FUNCTION_BLOCK Physical_Plant_SIMULATION (* Composite Function Block Type *)
  (* Standard: 61499-2 *)
  (* Version 0.0, 12/12/2023, Cheyan, Schneider Electric, template *)
  PACKAGE Main;
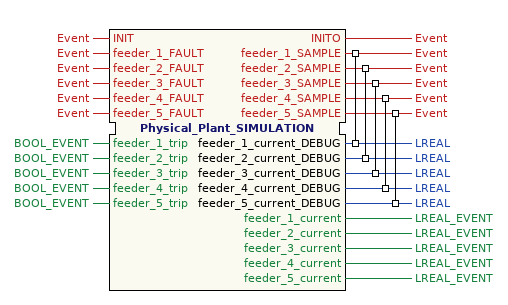
  EVENT_INPUT
    INIT; (* Initialization Request *)
    feeder_1_FAULT;
    feeder_2_FAULT;
    feeder_3_FAULT;
    feeder_4_FAULT;
    feeder_5_FAULT;
  END_EVENT
  EVENT_OUTPUT
    INITO; (* Initialization Confirm *)
    feeder_1_SAMPLE WITH feeder_1_current_DEBUG;
    feeder_2_SAMPLE WITH feeder_2_current_DEBUG;
    feeder_3_SAMPLE WITH feeder_3_current_DEBUG;
    feeder_4_SAMPLE WITH feeder_4_current_DEBUG;
    feeder_5_SAMPLE WITH feeder_5_current_DEBUG;
  END_EVENT
  VAR_OUTPUT
    feeder_1_current_DEBUG : LREAL; (* Output event qualifier *)
    feeder_2_current_DEBUG : LREAL; (* Output event qualifier *)
    feeder_3_current_DEBUG : LREAL; (* Output event qualifier *)
    feeder_4_current_DEBUG : LREAL; (* Output event qualifier *)
    feeder_5_current_DEBUG : LREAL; (* Output event qualifier *)
  END_VAR
  SOCKETS
    feeder_1_trip : BOOL_EVENT;
    feeder_2_trip : BOOL_EVENT;
    feeder_3_trip : BOOL_EVENT;
    feeder_4_trip : BOOL_EVENT;
    feeder_5_trip : BOOL_EVENT;
  END_SOCKETS
  PLUGS
    feeder_1_current : LREAL_EVENT;
    feeder_2_current : LREAL_EVENT;
    feeder_3_current : LREAL_EVENT;
    feeder_4_current : LREAL_EVENT;
    feeder_5_current : LREAL_EVENT;
  END_PLUGS
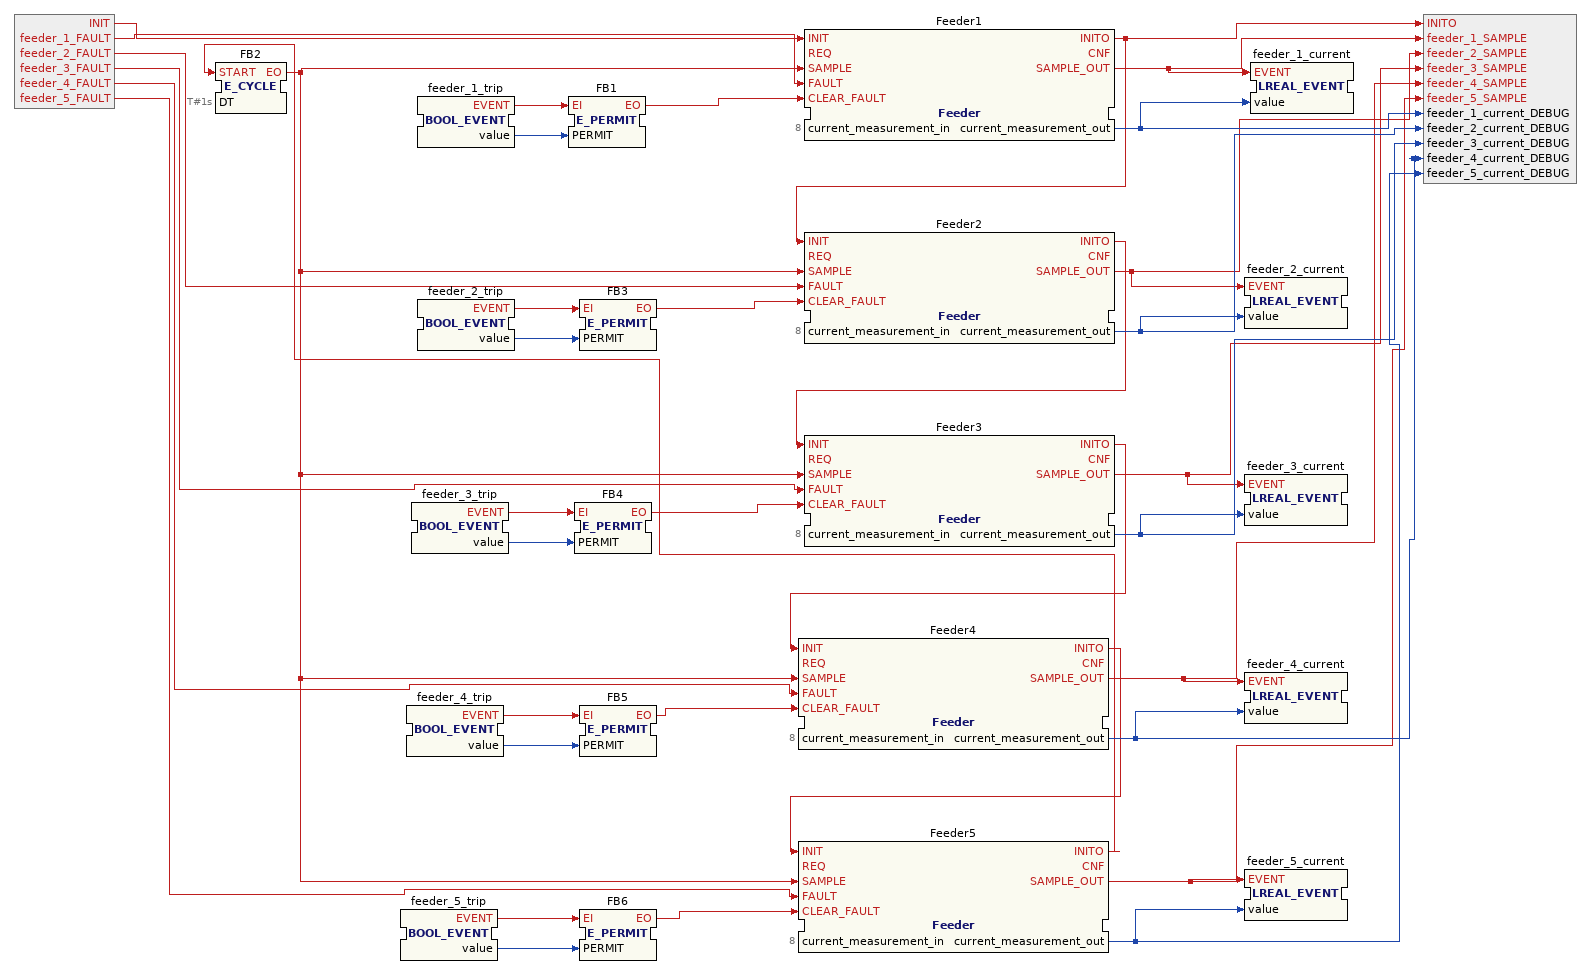
  FBS
    Feeder1 : Feeder(current_measurement_in := 8);
    FB2 : E_CYCLE(DT := T#1s);
    Feeder2 : Feeder(current_measurement_in := 8);
    Feeder3 : Feeder(current_measurement_in := 8);
    Feeder4 : Feeder(current_measurement_in := 8);
    Feeder5 : Feeder(current_measurement_in := 8);
    FB1 : E_PERMIT;
    FB3 : E_PERMIT;
    FB4 : E_PERMIT;
    FB5 : E_PERMIT;
    FB6 : E_PERMIT;
  END_FBS
  EVENT_CONNECTIONS
    FB2.EO TO Feeder1.SAMPLE;
    INIT TO Feeder1.INIT;
    Feeder1.INITO TO Feeder2.INIT;
    Feeder2.INITO TO Feeder3.INIT;
    Feeder3.INITO TO Feeder4.INIT;
    Feeder4.INITO TO Feeder5.INIT;
    Feeder5.INITO TO FB2.START;
    feeder_1_FAULT TO Feeder1.FAULT;
    feeder_2_FAULT TO Feeder2.FAULT;
    FB2.EO TO Feeder2.SAMPLE;
    FB2.EO TO Feeder3.SAMPLE;
    feeder_3_FAULT TO Feeder3.FAULT;
    feeder_4_FAULT TO Feeder4.FAULT;
    FB2.EO TO Feeder4.SAMPLE;
    FB2.EO TO Feeder5.SAMPLE;
    feeder_5_FAULT TO Feeder5.FAULT;
    Feeder1.SAMPLE_OUT TO feeder_1_SAMPLE;
    Feeder1.INITO TO INITO;
    Feeder2.SAMPLE_OUT TO feeder_2_SAMPLE;
    Feeder3.SAMPLE_OUT TO feeder_3_SAMPLE;
    Feeder4.SAMPLE_OUT TO feeder_4_SAMPLE;
    Feeder5.SAMPLE_OUT TO feeder_5_SAMPLE;
    Feeder1.SAMPLE_OUT TO feeder_1_current.EVENT;
    Feeder2.SAMPLE_OUT TO feeder_2_current.EVENT;
    Feeder3.SAMPLE_OUT TO feeder_3_current.EVENT;
    Feeder4.SAMPLE_OUT TO feeder_4_current.EVENT;
    Feeder5.SAMPLE_OUT TO feeder_5_current.EVENT;
    feeder_1_trip.EVENT TO FB1.EI;
    FB1.EO TO Feeder1.CLEAR_FAULT;
    feeder_2_trip.EVENT TO FB3.EI;
    FB3.EO TO Feeder2.CLEAR_FAULT;
    feeder_3_trip.EVENT TO FB4.EI;
    FB4.EO TO Feeder3.CLEAR_FAULT;
    feeder_4_trip.EVENT TO FB5.EI;
    FB5.EO TO Feeder4.CLEAR_FAULT;
    feeder_5_trip.EVENT TO FB6.EI;
    FB6.EO TO Feeder5.CLEAR_FAULT;
  END_CONNECTIONS
  DATA_CONNECTIONS
    Feeder1.current_measurement_out TO feeder_1_current_DEBUG;
    Feeder2.current_measurement_out TO feeder_2_current_DEBUG;
    Feeder3.current_measurement_out TO feeder_3_current_DEBUG;
    Feeder4.current_measurement_out TO feeder_4_current_DEBUG;
    Feeder5.current_measurement_out TO feeder_5_current_DEBUG;
    Feeder1.current_measurement_out TO feeder_1_current.value;
    Feeder2.current_measurement_out TO feeder_2_current.value;
    Feeder3.current_measurement_out TO feeder_3_current.value;
    Feeder4.current_measurement_out TO feeder_4_current.value;
    Feeder5.current_measurement_out TO feeder_5_current.value;
    feeder_1_trip.value TO FB1.PERMIT;
    feeder_2_trip.value TO FB3.PERMIT;
    feeder_3_trip.value TO FB4.PERMIT;
    feeder_4_trip.value TO FB5.PERMIT;
    feeder_5_trip.value TO FB6.PERMIT;
  END_CONNECTIONS
END_FUNCTION_BLOCK
